TYPE udt_ECATSlave_Status_EP9128 :
	STRUCT
		State: UINT;
		(*
		0x___1 = Slave in 'INIT' state
		0x___2 = Slave in 'PREOP' state
		0x___3 = Slave in 'BOOT' state
		0x___4 = Slave in 'SAFEOP' state
		0x___8 = Slave in 'OP' state
		0x001_ = Slave signals error
		0x002_ = Invalid vendorId, productCode... read
		0x004_ = Initialization error occurred
		0x008_ = Slave disabled
		0x010_ = Slave NOT present
		0x020_ = Slave signals link error
		0x040_ = Slave signals missing link
		0x080_ = Slave signals unexpected link
		0x100_ = Communication port A
		0x200_ = Communication port B
		0x400_ = Communication port C
		0x800_ = Communication port D
		*)
	END_STRUCT
END_TYPE

(* stored: Version 1.1.0.1, ProductVersion 3.1.4024.12
   DUT udt_ECATSlave_Status_EP9128: Id {1af4ca56-118a-4024-a21e-3365ad8a57de} *)
